FUNCTION_BLOCK FB_homeToSensorCustom
VAR_IN_OUT
	Axis : AXIS_REF;					
END_VAR
VAR_INPUT
	Execute 		: BOOL;
	Direction 		: INT; // 0- PositiveDirection, 1- NegativeDirection
	Velocity 		: LREAL;
	Acceleration 	: LREAL;
	Deceleration 	: LREAL;
	SetPosition 	: LREAL;
	TimeLimit 		: TIME;
	TorqueLimit 	: LREAL;
	BackOffPos 		: LREAL;
	homeSensor		: BOOL;
END_VAR
VAR_OUTPUT
	Done 			: BOOL;
	Busy 			: BOOL;
	Active 			: BOOL;
	CommandAborted 	: BOOL;
	Error 			: BOOL;
	ErrorID 		: UDINT;
END_VAR
VAR
	nState 			: INT;
	fbExecute 		: R_TRIG;
	fbTimeout 		: TON;
	fbDetectTime 	: TON;
	
	readParameter 		: MC_ReadParameter;
	readParameterOut 	: ST_mcOutputs;
	
	writeParameter		: MC_WriteParameter;
	writeParameterOut 	: ST_mcOutputs;
	readValue 			: LREAL;
	
	parameter 	: MC_AxisParameter;	
	writeValue 	: LREAL;
	
	moveToTorque	: MC_TorqueControl;
	torqueOptions 	: ST_TorqueControlOptions;
	moveToTorqueOut : ST_mcOutputs;
	
	moveAbsolute	: MC_MoveAbsolute;
	moveAbsoluteOut : ST_mcOutputs;
	calcBackOffPos 	: LREAL;
	
	home	: MC_Home;
	homeOut : ST_mcOutputs;
	
	stop		: MC_Stop;
	stopOut 	: ST_mcOutputs;
	fPosition	: LREAL;

	jog		: MC_Jog;
	jogOut 	: ST_mcOutputs;
	
	moveRelative	: MC_MoveRelative;
	moveRelativeOut	: ST_mcOutputs;
END_VAR

// Copy of FB_homeToTorque but torque homing indicator is replaced with a homing sensor connected to the motor class. 
//Similiar to homeToSensor() method found in motor class. This function works better with motors that are not inverted. (ie motors that gain positive counts when moving away from their home position).
//homeToSensor() uses built in beckhoff homing function and works well when motor is invereted. I could not find a way to switch the direction of the homing back off after sensor was found so I created
//this custom function that accomplishes the same thing. 

fbExecute(CLK := Execute);
fbTimeout();
actHome();
actMode();
actMove();


CASE nState OF 
	0: //init
		IF NOT Execute THEN
		(* reset at falling edge of Execute *)
			Busy 					:= FALSE;
			Done					:= FALSE;
			CommandAborted 			:= FALSE;
			Error 					:= FALSE;
			ErrorID 				:= 0;
			fbTimeout.IN 			:= FALSE;
			readParameter.Enable 	:= FALSE;
			writeParameter.Execute	:= FALSE;
			stop.Execute		 	:= FALSE;
			home.Execute 			:= FALSE;
			moveAbsolute.Execute 	:= FALSE;
			jog.JogForward 			:= FALSE;
			jog.JogBackwards 		:= FALSE;
		END_IF
	
		IF fbExecute.Q THEN
			Busy := TRUE;
			nState := nState + 1;
		END_IF
		
	1:// Check homeSensor
		(*IF homeSensor THEN
			nState := 6;
		ELSE 
			nState := nState + 1;
		END_IF*)
		nState := nState + 1;
	2:// Read soft limit switch to set back to when done
		CASE Direction OF 
			0: //mcPositiveDirection
		      	parameter := AxisMaxSoftPosLimit;
			1: //mcNegativeDirection
				parameter := AxisMinSoftPosLimit;
		END_CASE
		
		readParameter.Enable := TRUE;
		
		IF NOT readParameterOut.Busy AND readParameterOut.Done THEN
			readParameter.Enable := FALSE;
			nState := nState + 1;
		ELSIF NOT readParameterOut.Busy AND readParameterOut.Error THEN
			Error := readParameterOut.Error;
			ErrorId := readParameterOut.ErrorID;
			readParameter.Enable := FALSE;
			nState := 0;
		END_IF
		
	3: // Set soft limit switch to appropriate allowance
		CASE Direction OF
			0 : //mcPositiveDirection
				writeValue := 99999;
			1 : //mcNegativeDirection
				writeValue := -99999;
		END_CASE
		
		writeParameter.Execute := TRUE;
		
		IF NOT writeParameterOut.Busy AND writeParameterOut.Done THEN
			writeParameter.Execute := FALSE;
			nState := nState + 1;
		ELSIF NOT writeParameterOut.Busy AND writeParameterOut.Error THEN
			Error := writeParameterOut.Error;
			ErrorID := writeParameterOut.ErrorID;
			writeParameter.Execute := FALSE;
			nState := 0;
		END_IF
		
	4: //Execute MoveTowards Sensor
		fbTimeout(IN:= TRUE, PT:= TimeLimit);
		
		CASE Direction OF
			0: //mcPositiveDirection 
				jog.JogForward := TRUE;
				jog.JogBackwards := FALSE;
			1: //mcNegativeDirection 
				jog.JogForward := FALSE;
				jog.JogBackwards := TRUE;
		END_CASE
			
		IF homeSensor THEN
			jog.JogForward := FALSE;
			jog.JogBackwards := FALSE;
			nState := nState + 1;
		ELSIF NOT jogOut.Busy AND jogOut.Error THEN
			Error := jogOut.Error;
			ErrorID := jogOut.ErrorID;
			jog.JogForward := FALSE;
			jog.JogBackwards := FALSE;
			nState := 0;
		END_IF
		
		// Timeout Error
		IF fbTimeout.Q THEN
			jog.JogForward := FALSE;
			jog.JogBackwards := FALSE;
			Error := TRUE;
			ErrorID := 1;
			nState := 0;
		END_IF
		
		CommandAborted := jogOut.CommandAborted;
		
	5://Stop motor 
		stop.Execute := TRUE;
		
		IF stopOut.Busy AND stopOut.Done THEN
			stop.Execute := FALSE;
			CASE Direction OF
				0: //mcPositiveDirection 
					calcBackOffPos := -BackOffPos;
				1: //mcNegativeDirection 
					calcBackOffPos := BackOffPos;
			END_CASE
			nState := nState + 1;
			
		ELSIF NOT stopOut.Busy AND stopOut.Error THEN
			Error := stopOut.Error;
			ErrorId := stopOut.ErrorID;
			stop.Execute := FALSE;
			nState := 0;
		END_IF
		
		CommandAborted := stopOut.CommandAborted;
		
	7: //Set homing state and counts
		IF axis.status.StandStill THEN
			home.Execute := TRUE;
		END_IF
		
		IF NOT homeOut.Busy AND homeOut.Done THEN
			home.Execute := FALSE;
			nState := nState + 1;
		ELSIF NOT homeOut.Busy AND homeOut.Error THEN
			Error := homeOut.Error;
			ErrorId := homeOut.ErrorID;
			home.Execute := FALSE;
			nState := 0;
		END_IF
		
		CommandAborted := homeOut.CommandAborted;
		
	6: //Move off home slightly
		IF axis.status.StandStill THEN
			moveRelative.Execute := TRUE;
		END_IF
		
		IF NOT moveRelativeOut.Busy AND moveRelativeOut.Done THEN
			moveRelative.Execute := FALSE;
			nState := nState + 1;
		ELSIF NOT moveRelativeOut.Busy AND moveRelativeOut.Error THEN
			Error := moveRelativeOut.Error;
			ErrorId := moveRelativeOut.ErrorID;
			moveRelative.Execute := FALSE;
			nState := 0;
		END_IF
		
		CommandAborted := moveRelativeOut.CommandAborted;
		
	8: // Write limit switch to original Value
		writeValue := SetPosition;
		writeParameter.Execute := TRUE;
		
		IF NOT writeParameterOut.Busy AND writeParameterOut.Done THEN
			writeParameter.Execute := FALSE;
			Busy := FALSE;
			Done := TRUE;
			nState := 0;
		ELSIF NOT writeParameterOut.Busy AND writeParameterOut.Error THEN
			Error := writeParameterOut.Error;
			ErrorID := writeParameterOut.ErrorID;
			writeParameter.Execute := FALSE;
			nState := 0;
		END_IF
END_CASE

IF axis.Status.Error THEN
	nState := 0;
END_IF

ACTION actHome:
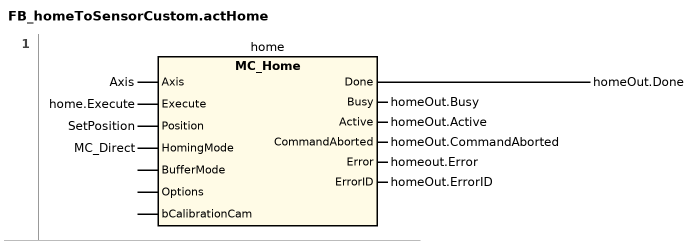
// NETWORK 1
home(
    Axis := Axis,
    Execute := home.Execute,
    Position := SetPosition,
    HomingMode := MC_Direct,
    Busy => homeOut.Busy,
    Active => homeOut.Active,
    CommandAborted => homeOut.CommandAborted,
    Error => homeout.Error,
    ErrorID => homeOut.ErrorID); // MC_Home
homeOut.Done := home.Done;
END_ACTION

ACTION actMode:
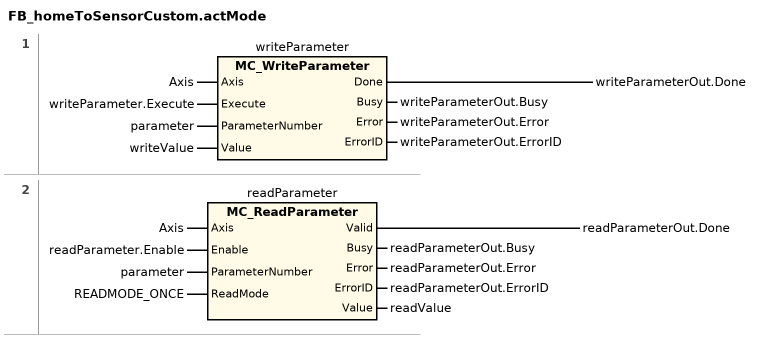
// NETWORK 1
writeParameter(
    Axis := Axis,
    Execute := writeParameter.Execute,
    ParameterNumber := parameter,
    Value := writeValue,
    Busy => writeParameterOut.Busy,
    Error => writeParameterOut.Error,
    ErrorID => writeParameterOut.ErrorID); // MC_WriteParameter
writeParameterOut.Done := writeParameter.Done;

// NETWORK 2
readParameter(
    Axis := Axis,
    Enable := readParameter.Enable,
    ParameterNumber := parameter,
    ReadMode := READMODE_ONCE,
    Busy => readParameterOut.Busy,
    Error => readParameterOut.Error,
    ErrorID => readParameterOut.ErrorID,
    Value => readValue); // MC_ReadParameter
readParameterOut.Done := readParameter.Valid;
END_ACTION

ACTION actMove:
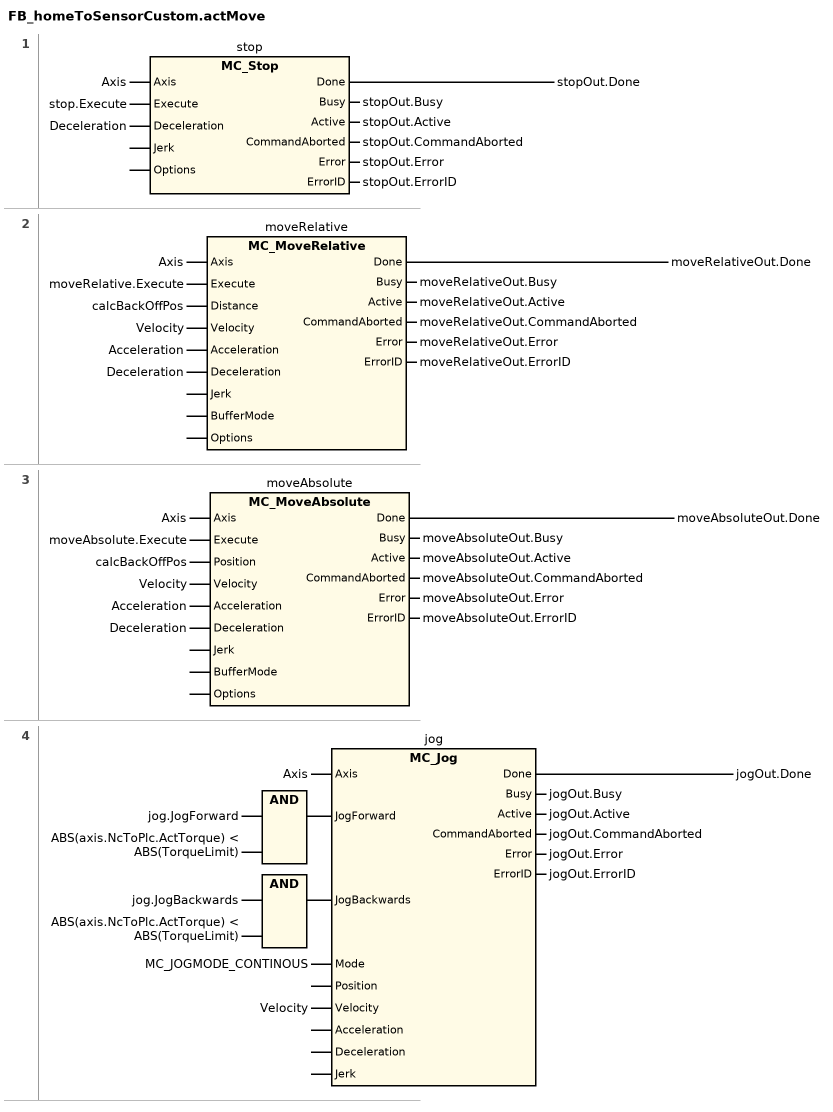
// NETWORK 1
stop(
    Axis := Axis,
    Execute := stop.Execute,
    Deceleration := Deceleration,
    Busy => stopOut.Busy,
    Active => stopOut.Active,
    CommandAborted => stopOut.CommandAborted,
    Error => stopOut.Error,
    ErrorID => stopOut.ErrorID); // MC_Stop
stopOut.Done := stop.Done;

// NETWORK 2
moveRelative(
    Axis := Axis,
    Execute := moveRelative.Execute,
    Distance := calcBackOffPos,
    Velocity := Velocity,
    Acceleration := Acceleration,
    Deceleration := Deceleration,
    Busy => moveRelativeOut.Busy,
    Active => moveRelativeOut.Active,
    CommandAborted => moveRelativeOut.CommandAborted,
    Error => moveRelativeOut.Error,
    ErrorID => moveRelativeOut.ErrorID); // MC_MoveRelative
moveRelativeOut.Done := moveRelative.Done;

// NETWORK 3
moveAbsolute(
    Axis := Axis,
    Execute := moveAbsolute.Execute,
    Position := calcBackOffPos,
    Velocity := Velocity,
    Acceleration := Acceleration,
    Deceleration := Deceleration,
    Busy => moveAbsoluteOut.Busy,
    Active => moveAbsoluteOut.Active,
    CommandAborted => moveAbsoluteOut.CommandAborted,
    Error => moveAbsoluteOut.Error,
    ErrorID => moveAbsoluteOut.ErrorID); // MC_MoveAbsolute
moveAbsoluteOut.Done := moveAbsolute.Done;

// NETWORK 4
jog(
    Axis := Axis,
    JogForward := jog.JogForward AND (ABS(axis.NcToPlc.ActTorque) < ABS(TorqueLimit)),
    JogBackwards := jog.JogBackwards AND (ABS(axis.NcToPlc.ActTorque) < ABS(TorqueLimit)),
    Mode := MC_JOGMODE_CONTINOUS,
    Velocity := Velocity,
    Busy => jogOut.Busy,
    Active => jogOut.Active,
    CommandAborted => jogOut.CommandAborted,
    Error => jogOut.Error,
    ErrorID => jogOut.ErrorID); // MC_Jog
jogOut.Done := jog.Done;
END_ACTION

END_FUNCTION_BLOCK

(* stored: Version 1.1.0.1, ProductVersion 3.1.4024.13
   POU FB_homeToSensorCustom: Id {d0a94e40-362a-4e54-9284-4a83812ac785}, SpecialFunc None
   Action actHome: Id {2a7de268-cd20-4e31-97c5-f419007108bd}
   Action actMode: Id {be23baa4-2aad-451f-bb00-09c55a43f769}
   Action actMove: Id {ffa759d6-f796-4c1c-b896-c9c2f523d25d} *)
